RoboDK station: Endelig robodk fremvisning.rdk

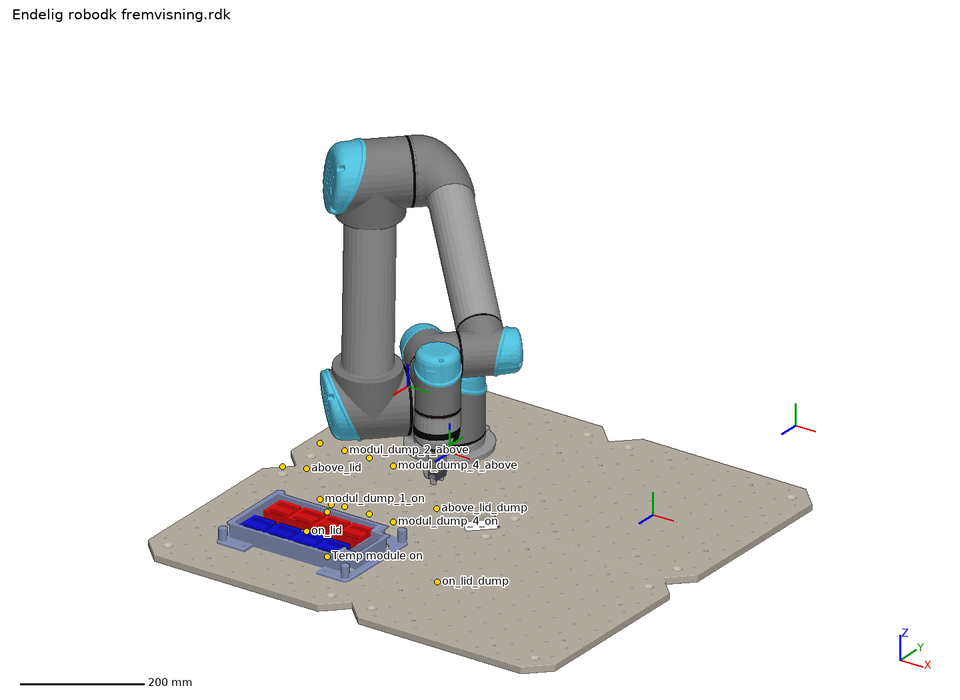
[picture v0: the station drawn from its stored meshes, robots at their saved joint values, targets as dots, program paths as lines]
Station Endelig robodk fremvisning (saved by RoboDK 6.0.3). Poses are relative to the parent item; angles as X-Y-Z fixed-axis rotations.
  - frame World frame at (-180, 140, 0) mm, rotated rx 0 ry 0 rz -90 deg
    - object Battery_chasis_assembly_214 (1) at (480, 80, 0) mm, size 180.1 x 260 x 34 mm, geometry from Battery_chasis_assembly_214 (1).STEP
    - object BMW red module  at (526, 122, 0) mm, size 42 x 48 x 26 mm, geometry from 003_BMW_Module_STEP.stp
    - object BMW red module at (526, 180, 0.3) mm, size 42 x 48 x 26 mm, geometry from 003_BMW_Module_STEP.stp
    - object BMW red module at (526, 218, -0.14) mm, size 42 x 48 x 26 mm, geometry from 003_BMW_Module_STEP.stp
    - object BMW red module at (526, 266, -0.14) mm, size 42 x 48 x 26 mm, geometry from 003_BMW_Module_STEP.stp
    - object BMW blue module  at (595, 120, 0) mm, size 42 x 48 x 26 mm, geometry from 003_BMW_Module_STEP.stp
    - object BMW blue module  at (595, 170, 0) mm, size 42 x 48 x 26 mm, geometry from 003_BMW_Module_STEP.stp
    - object BMW blue module  at (595, 218, 0) mm, size 42 x 48 x 26 mm, geometry from 003_BMW_Module_STEP.stp
    - object BMW blue module  at (595, 266, 0) mm, size 42 x 48 x 26 mm, geometry from 003_BMW_Module_STEP.stp
    - object 002_BMW_Battery_Lid_ STEP_Colour at (560, 194, 1031) mm, size 140 x 244 x 7 mm, geometry from 002_BMW_Battery_Lid_ STEP_Colour.STEP
    - target above_lid (Cartesian target) at (560, 194, 131) mm, rotated rx 180 ry 0 rz -180 deg; joints [-72.817, -85.214, -123.022, -61.779, 89.799, 107.064] of UR5
    - target on_lid (Cartesian target) at (560, 194, 18) mm, rotated rx 180 ry 0 rz 180 deg; joints [-72.812, -93.5, -130.041, -46.473, 89.818, 107.018] of UR5
    - target above_lid_dump (Cartesian target) at (560.1, 449.51, 130.93) mm, rotated rx 179.98 ry -0.01 rz -90.13 deg; joints [-44.49, -96.139, -111.952, -61.942, 89.824, 45.517] of UR5
    - target on_lid_dump (Cartesian target) at (560, 450, 0) mm, rotated rx -180 ry 0 rz -90 deg; joints [-44.43, -108.468, -120.561, -40.985, 89.85, 45.376] of UR5
    - target module_position_FIRST (Cartesian target) at (595, 266, 100) mm, rotated rx 180 ry 0 rz -90.14 deg; joints [-65.453, -93.745, -119.869, -56.403, 89.813, 24.542] of UR5
    - target module_position_SECOND (Cartesian target) at (526, 122, 100) mm, rotated rx 180 ry 0 rz -90.14 deg; joints [-82.076, -83.399, -129.875, -56.743, 89.796, 7.93] of UR5
    - target modul_dump_4_above (Cartesian target) at (420, 266, 100) mm, rotated rx 180 ry 0 rz -90.14 deg; joints [-50.776, -66.181, -141.434, -62.402, 89.772, 39.27] of UR5
    - target modul_dump_4_on (Cartesian target) at (420, 266, 0) mm, rotated rx 180 ry 0 rz -90.14 deg; joints [-50.762, -82.003, -151.129, -36.885, 89.807, 39.191] of UR5
    - target modul_dump_3_above (Cartesian target) at (420, 218, 100) mm, rotated rx 180 ry 0 rz -90.14 deg; joints [-59.27, -63.997, -142.5, -63.521, 89.77, 30.782] of UR5
    - target modul_dump_3_on (Cartesian target) at (420, 218, 0) mm, rotated rx 180 ry 0 rz -90.14 deg; joints [-59.256, -80.071, -152.52, -37.426, 89.804, 30.701] of UR5
    - target modul_dump_2_above (Cartesian target) at (420, 170, 100) mm, rotated rx 180 ry 0 rz -90.14 deg; joints [-68.838, -63.48, -142.74, -63.797, 89.769, 21.216] of UR5
    - target modul_dump_2_on (Cartesian target) at (420, 170, 0) mm, rotated rx 180 ry 0 rz -90.14 deg; joints [-68.823, -79.606, -152.839, -37.572, 89.802, 21.135] of UR5
    - target modul_dump_1_above (Cartesian target) at (420, 122, 100) mm, rotated rx 180 ry 0 rz -90.14 deg; joints [-78.986, -64.719, -142.156, -63.141, 89.77, 11.063] of UR5
    - target modul_dump_1_on (Cartesian target) at (420, 122, 0) mm, rotated rx 180 ry 0 rz -90.14 deg; joints [-78.972, -80.715, -152.068, -37.233, 89.804, 10.984] of UR5
    - target Temp module move above (Cartesian target) at (595.83, 258.8, 85) mm, rotated rx 180 ry 0 rz -90.14 deg; joints [-65.453, -93.745, -119.869, -56.403, 89.813, 24.542] of UR5
    - target Temp module above (Cartesian target) at (595.83, 258.8, 85) mm, rotated rx 180 ry 0 rz -90.14 deg; joints [-65.453, -93.745, -119.869, -56.403, 89.813, 24.542] of UR5
    - target Temp module on (Cartesian target) at (595.83, 258.8, 5) mm, rotated rx 180 ry 0 rz -90.14 deg; joints [-65.453, -93.745, -119.869, -56.403, 89.813, 24.542] of UR5
  - frame UR5 Base at (0, 0, 0) mm
    - robot UR5: 6 axes
        modified DH rows (alpha deg, a mm, theta deg, d mm): 0, 0, 0, 89.2; 90, 0, 180, 0; 0, 425, 0, 0; 0, 392, 0, 109.3; -90, 0, 0, 94.75; 90, 0, 180, 82.5
        joint limits [-360, -360, -360, -360, -360, -360] to [360, 360, 360, 360, 360, 360]; home [0, -90, -90, 0, 90, 0]; saved at [-44.499, -94.287, -109.296, -66.467, 89.814, 45.503]
      - tool Mecademic SCHUNK MPG-plus 25 Gripper (Closed), TCP at (0, 0, 142) mm, size 70.2 x 49.2 x 28.5 mm
      - tool AdapterUR5_v3, TCP at (0, 0, 200) mm, size 75 x 75 x 35.2 mm, geometry from AdapterUR5_v3.STL
  - frame Frame 1 at (0, 0, -12) mm, rotated rx 90 ry 0 rz 0 deg
    - object plate0x0y at (0, 0, 0) mm, size 399.5 x 12 x 399.5 mm, geometry from pallette_1x1-perforated_m6-ahl-001.STEP
  - frame Frame 2 at (400, 0, -12) mm, rotated rx 90 ry 0 rz 0 deg
    - object plate1x0y at (0, 0, 0) mm, size 399.5 x 12 x 399.5 mm, geometry from pallette_1x1-perforated_m6-ahl-001.STEP
  - frame Frame 4 at (400, 400, -12) mm, rotated rx 90 ry 0 rz 0 deg
    - object plate1x1y at (0, 0, 800) mm, size 399.5 x 12 x 399.5 mm, geometry from pallette_1x1-perforated_m6-ahl-001.STEP
  - program P240Battery (76 instructions, listed below)
  - object plate1x0y at (0, -400, -12) mm, rotated rx 90 ry 0 rz 0 deg, size 399.5 x 12 x 399.5 mm, geometry from pallette_1x1-perforated_m6-ahl-001.STEP
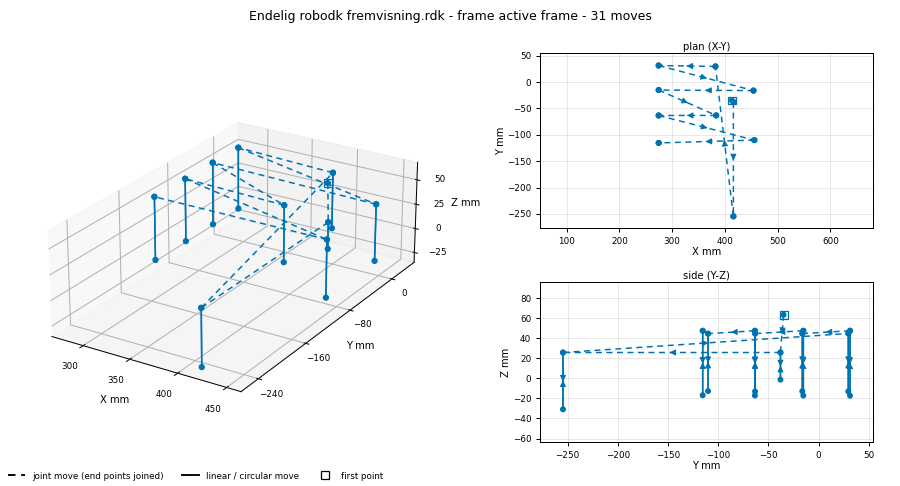
[picture p0: tool path of Endelig robodk fremvisning.rdk in frame active frame, 31 of 31 moves have a stored position in this frame; points joined in program order, loops and branches not executed]

--- program P240Battery (robot UR5) ---
  step_count_32f61c6e_5ec4_4497_8514_23adf8940269 = 0.0
  Call thread Step_Counter_Thread_d25f110d_83c6_4cc4_90fa_39eb4fdbfc4f:
  while (True):
  step_count_32f61c6e_5ec4_4497_8514_23adf8940269 = step_count_32f61c6e_5ec4_4497_8514_23adf8940269 + 1.0
  Call sync
  end
  end
  Call run Step_Counter_Thread_d25f110d_83c6_4cc4_90fa_39eb4fdbfc4f
  Call set_standard_analog_input_domain(0, 1)
  Call set_standard_analog_input_domain(1, 1)
  Call set_tool_analog_input_domain(0, 1)
  Call set_tool_analog_input_domain(1, 1)
  Call set_analog_outputdomain(0, 0)
  Call set_analog_outputdomain(1, 0)
  Call set_input_actions_to_default
  Call set_safety_mode_transition_hardness(1)
  Set Tool at (0, 0, 150) mm
  Call set_payload(0.25)
  Call set_tool_voltage(0)
  Call set_gravity([0.0, 0.0, 9.82])
  global i_var_1=1
  while (True):
  MoveJ to (413.19, -34.88, 63.27) mm, rotated rx 180 ry 1 rz -90 deg; joints [10.084, -87.084, -126.597, -56.164, 90.792, 9.949]
  MoveJ to (416.11, -37.96, 25.72) mm, rotated rx -180 ry 0 rz -90 deg; joints [10.153, -91.329, -129.256, -49.426, 89.813, 9.99]
  Call set_standard_digital_out(6, True)
  Call set_standard_digital_out(7, False)
  MoveL to (416.14, -37.96, -1.34) mm, rotated rx -179.99 ry 0 rz -89.99 deg; joints [10.156, -94.606, -131.15, -44.25, 89.82, 9.97]
  Call set_standard_digital_out(7, True)
  Call set_standard_digital_out(6, False)
  MoveL to (416.11, -37.96, 25.72) mm, rotated rx -180 ry 0 rz -90 deg; joints [10.153, -91.329, -129.256, -49.426, 89.813, 9.99]
  MoveJ to (416.08, -254.66, 25.68) mm, rotated rx -180 ry 0.01 rz 0 deg; joints [-18.334, -100.36, -118.939, -50.724, 89.829, -108.496]
  MoveL to (416.12, -254.63, -30.9) mm, rotated rx -180 ry 0 rz 0 deg; joints [-18.327, -106.522, -122.114, -41.38, 89.848, -108.522]
  Call set_standard_digital_out(6, True)
  Call set_standard_digital_out(7, False)
  MoveL to (416.08, -254.66, 25.68) mm, rotated rx -180 ry 0.01 rz 0 deg; joints [-18.334, -100.36, -118.939, -50.724, 89.829, -108.496]
  MoveJ to (382.08, 29.64, 44.67) mm, rotated rx 180 ry 0 rz 0 deg; joints [21.174, -108.364, -104.845, 123.217, -89.837, 111.078]
  MoveL to (382.06, 29.6, -13.05) mm, rotated rx 180 ry 0.01 rz 0 deg; joints [21.161, -113.299, -108.13, 131.426, -89.851, 111.042]
  Call set_standard_digital_out(7, True)
  Call set_standard_digital_out(6, False)
  MoveL to (382.08, 29.64, 44.67) mm, rotated rx 180 ry 0 rz 0 deg; joints [21.174, -108.364, -104.845, 123.217, -89.837, 111.078]
  MoveJ to (274.4, 31.35, 47.42) mm, rotated rx -179.99 ry 0.01 rz 0.01 deg; joints [30.02, -94.374, -121.965, 126.34, -89.825, 119.913]
  MoveL to (274.42, 31.34, -17.28) mm, rotated rx -180 ry 0.01 rz 0.01 deg; joints [29.997, -101.446, -126.207, 137.654, -89.842, 119.858]
  Call set_standard_digital_out(6, True)
  Call set_standard_digital_out(7, False)
  MoveL to (274.4, 31.35, 47.42) mm, rotated rx -179.99 ry 0.01 rz 0.01 deg; joints [30.02, -94.374, -121.965, 126.34, -89.825, 119.913]
  MoveJ to (454.24, -16.18, 44.54) mm, rotated rx -179.99 ry 0.02 rz 0.02 deg; joints [12.021, -117.019, -92.006, 119.017, -89.87, 101.913]
  MoveL to (454.19, -16.23, -12.81) mm, rotated rx -180 ry 0.02 rz -0.01 deg; joints [12.063, -121.114, -95.282, 126.358, -89.839, 101.888]
  Call set_standard_digital_out(7, True)
  Call set_standard_digital_out(6, False)
  MoveL to (454.24, -16.18, 44.54) mm, rotated rx -179.99 ry 0.02 rz 0.02 deg; joints [12.021, -117.019, -92.006, 119.017, -89.87, 101.913]
  MoveJ to (274.39, -15.17, 47.41) mm, rotated rx -179.99 ry 0.01 rz 0.01 deg; joints [20.463, -94.184, -122.177, 126.359, -89.824, 110.36]
  MoveL to (274.41, -15.18, -17.17) mm, rotated rx -179.99 ry 0.01 rz 0 deg; joints [20.439, -101.264, -126.423, 137.685, -89.844, 110.303]
  Call set_standard_digital_out(6, True)
  Call set_standard_digital_out(7, False)
  MoveL to (274.39, -15.17, 47.41) mm, rotated rx -179.99 ry 0.01 rz 0.01 deg; joints [20.463, -94.184, -122.177, 126.359, -89.824, 110.36]
  MoveJ to (383.52, -63.26, 44.6) mm, rotated rx 180 ry 0 rz 0.02 deg; joints [7.132, -109.037, -103.908, 122.95, -89.838, 97.018]
  MoveL to (383.5, -63.28, -13.03) mm, rotated rx 180 ry 0 rz 0.02 deg; joints [7.122, -113.902, -107.173, 131.079, -89.85, 96.985]
  Call set_standard_digital_out(7, True)
  Call set_standard_digital_out(6, False)
  MoveL to (383.52, -63.26, 44.6) mm, rotated rx 180 ry 0 rz 0.02 deg; joints [7.132, -109.037, -103.908, 122.95, -89.838, 97.018]
  MoveJ to (274.4, -63.4, 47.4) mm, rotated rx -179.99 ry 0.01 rz 0.01 deg; joints [10.016, -95.132, -121.128, 126.259, -89.823, 99.913]
  MoveL to (274.44, -63.41, -17.12) mm, rotated rx -179.99 ry 0 rz 0 deg; joints [9.994, -102.089, -125.316, 137.41, -89.843, 99.86]
  Call set_standard_digital_out(6, True)
  Call set_standard_digital_out(7, False)
  MoveL to (274.4, -63.4, 47.4) mm, rotated rx -179.99 ry 0.01 rz 0.01 deg; joints [10.016, -95.132, -121.128, 126.259, -89.823, 99.913]
  MoveJ to (455.88, -110.1, 44.5) mm, rotated rx -179.99 ry -0.12 rz -0.17 deg; joints [0.045, -118.706, -89.319, 118.151, -89.872, 90.13]
  MoveL to (455.87, -110.08, -12.75) mm, rotated rx -179.99 ry -0.12 rz -0.17 deg; joints [0.092, -102.222, -124.239, -43.436, 89.844, -89.926]
  Call set_standard_digital_out(7, True)
  Call set_standard_digital_out(6, False)
  MoveL to (455.88, -110.1, 44.5) mm, rotated rx -179.99 ry -0.12 rz -0.17 deg; joints [0.045, -118.706, -89.319, 118.151, -89.872, 90.13]
  MoveJ to (274.42, -115.44, 47.4) mm, rotated rx -180 ry 0.01 rz 0 deg; joints [-1.09, -97.316, -118.628, 125.944, -89.824, 88.812]
  MoveL to (274.43, -115.43, -16.88) mm, rotated rx -180 ry 0 rz 0 deg; joints [135.534, -76.066, 122.808, 43.249, 89.985, 45.262]
  Call set_standard_digital_out(6, True)
  Call set_standard_digital_out(7, False)
  MoveL to (274.42, -115.44, 47.4) mm, rotated rx -180 ry 0.01 rz 0 deg; joints [-1.09, -97.316, -118.628, 125.944, -89.824, 88.812]
  end
